// Mitsubishi GX Works2 project: test_485   PLC: FX3U/FX3UC

PROGRAM MAIN
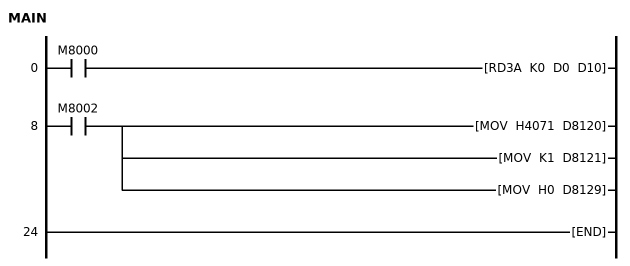
0     LD      M8000
      RD3A    K0 D0 D10
8     LD      M8002
      MOV     H4071 D8120
      MOV     K1 D8121
      MOV     H0 D8129
24    END
END_PROGRAM
